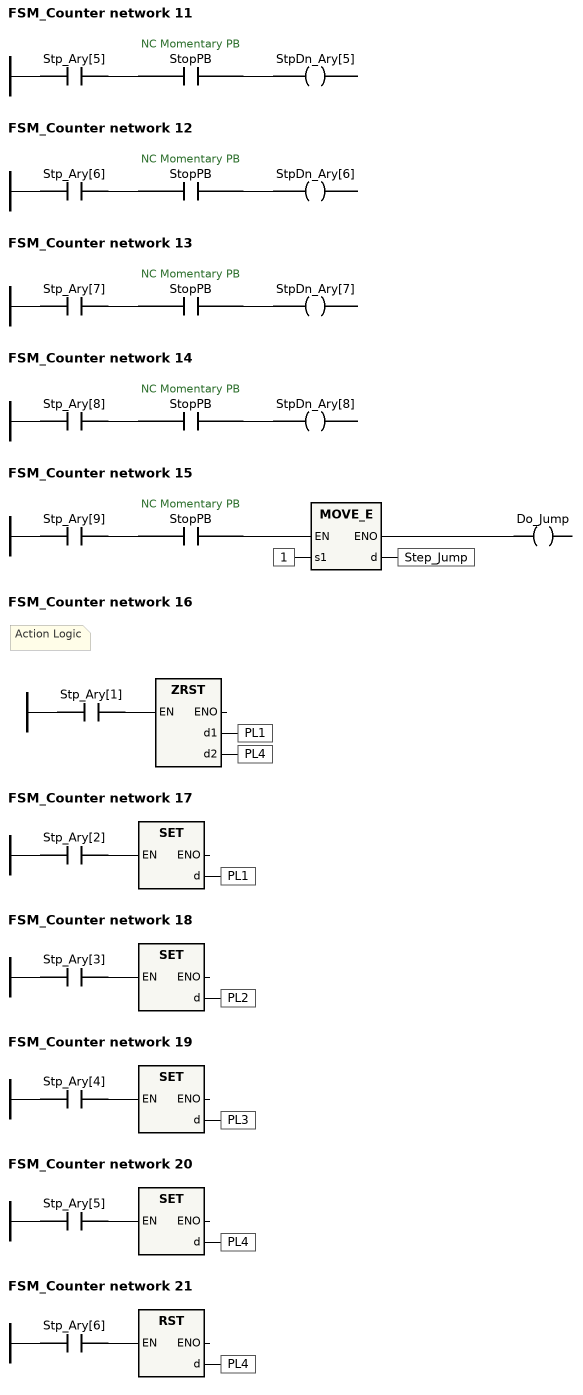
(* network 11 *)
StpDn_Ary[5] := Stp_Ary[5] AND StopPB;
(* network 12 *)
StpDn_Ary[6] := Stp_Ary[6] AND StopPB;
(* network 13 *)
StpDn_Ary[7] := Stp_Ary[7] AND StopPB;
(* network 14 *)
StpDn_Ary[8] := Stp_Ary[8] AND StopPB;
(* network 15 *)
_e1 := MOVE_E(Stp_Ary[9] AND StopPB, 1, Step_Jump);
Do_Jump := _e1;
(* network 16 *)
(* Action Logic *)
ZRST(Stp_Ary[1], PL1, PL4);
(* network 17 *)
SET(Stp_Ary[2], PL1);
(* network 18 *)
SET(Stp_Ary[3], PL2);
(* network 19 *)
SET(Stp_Ary[4], PL3);
(* network 20 *)
SET(Stp_Ary[5], PL4);
(* network 21 *)
RST(Stp_Ary[6], PL4);
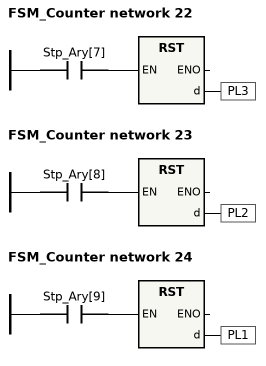
(* network 22 *)
RST(Stp_Ary[7], PL3);
(* network 23 *)
RST(Stp_Ary[8], PL2);
(* network 24 *)
RST(Stp_Ary[9], PL1);
END_PROGRAM

FUNCTION_BLOCK Get_Step_D
VAR_OUTPUT
  GSOut : BOOL;
END_VAR
VAR_IN_OUT
  SArray : ARRAY [0..15] OF BOOL;
END_VAR
VAR_INPUT
  StpNum : INT;
END_VAR
GSOut := SArray[StpNum];
END_FUNCTION_BLOCK

FUNCTION_BLOCK SR_Step_D
VAR_INPUT
  In : BOOL;
  StpNum : INT;
END_VAR
VAR_IN_OUT
  SArray : ARRAY [0..15] OF BOOL;
END_VAR
SArray[StpNum] := In;
END_FUNCTION_BLOCK

PROGRAM FSM_Counter_D
VAR
  StepCtrCV : INT;
  ClrStep : SR_Step;
  SetStep : SR_Step;
  Reset : BOOL;
  Do_Jump : BOOL;
  Step_Jump : INT;
  R_TRIG_1 : R_TRIG;
  Get_Step_D_1 : Get_Step_D;
  SR_Step_D_1 : SR_Step_D;
  SR_Step_D_2 : SR_Step_D;
END_VAR
(* structured ladder/FBD written out as ST: instructions are called as NAME(EN, inputs, outputs); _pN, _eN, _tN stand for wires *)
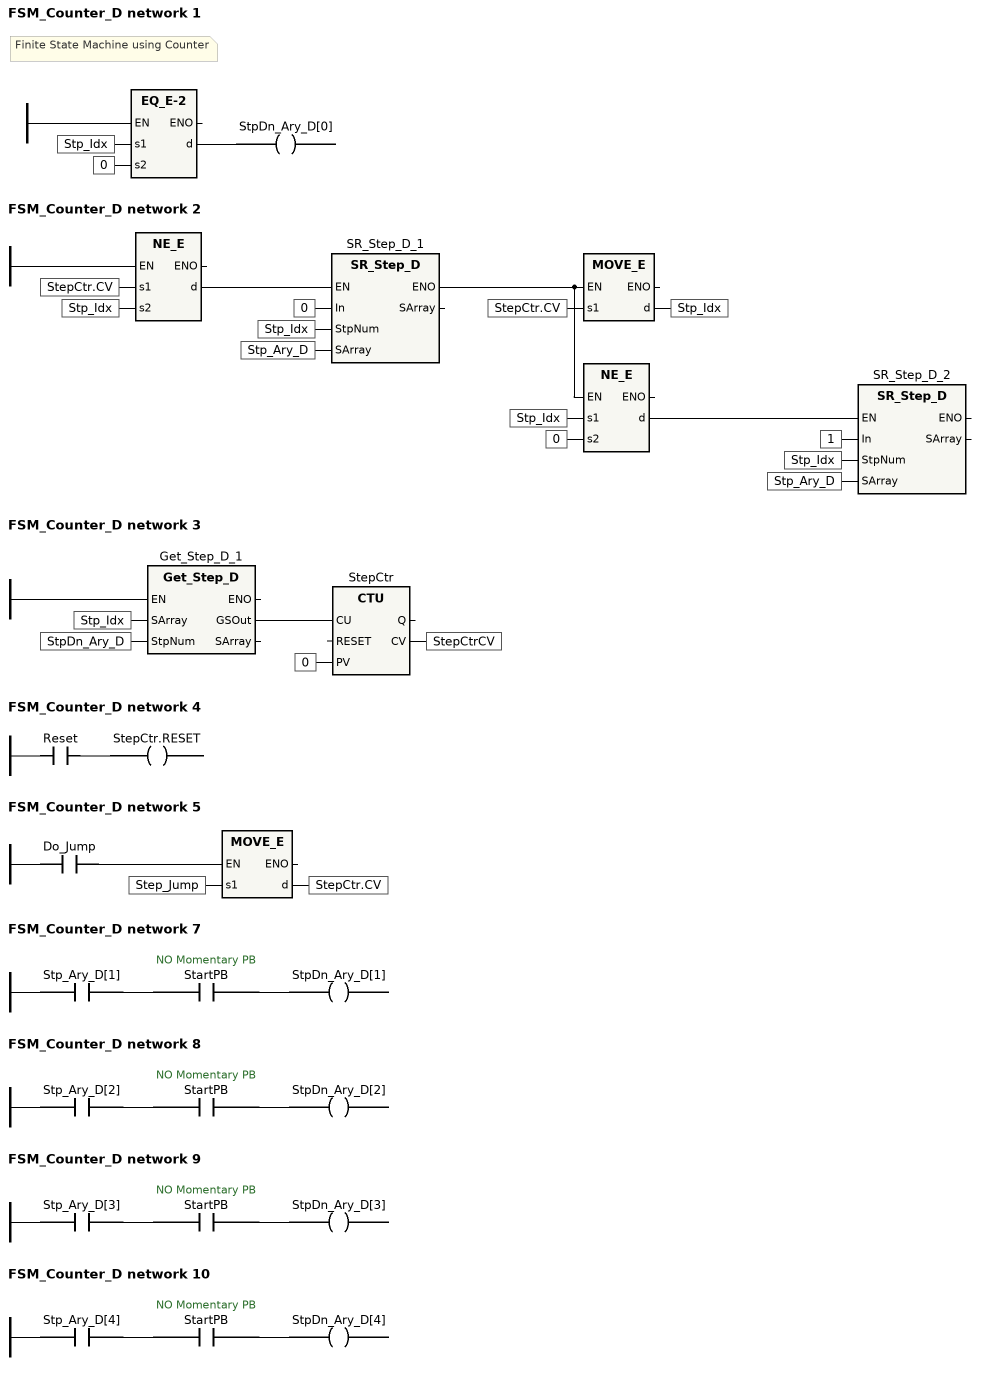
(* network 1 *)
(* Finite State Machine using Counter *)
EQ_E(TRUE, Stp_Idx, 0, _t1);
StpDn_Ary_D[0] := _t1;
(* network 2 *)
NE_E(TRUE, StepCtr.CV, Stp_Idx, _t1);
SR_Step_D_1(EN := _t1, In := 0, StpNum := Stp_Idx, SArray := Stp_Ary_D);
MOVE_E(SR_Step_D_1.ENO, StepCtr.CV, Stp_Idx);
NE_E(SR_Step_D_1.ENO, Stp_Idx, 0, _t2);
SR_Step_D_2(EN := _t2, In := 1, StpNum := Stp_Idx, SArray := Stp_Ary_D);
(* network 3 *)
Get_Step_D_1(EN := TRUE, SArray := Stp_Idx, StpNum := StpDn_Ary_D);
StepCtr(CU := Get_Step_D_1.GSOut, PV := 0, CV => StepCtrCV);
(* network 4 *)
StepCtr.RESET := Reset;
(* network 5 *)
MOVE_E(Do_Jump, Step_Jump, StepCtr.CV);
(* Transition Logic *)
(* network 7 *)
StpDn_Ary_D[1] := Stp_Ary_D[1] AND StartPB;
(* network 8 *)
StpDn_Ary_D[2] := Stp_Ary_D[2] AND StartPB;
(* network 9 *)
StpDn_Ary_D[3] := Stp_Ary_D[3] AND StartPB;
(* network 10 *)
StpDn_Ary_D[4] := Stp_Ary_D[4] AND StartPB;
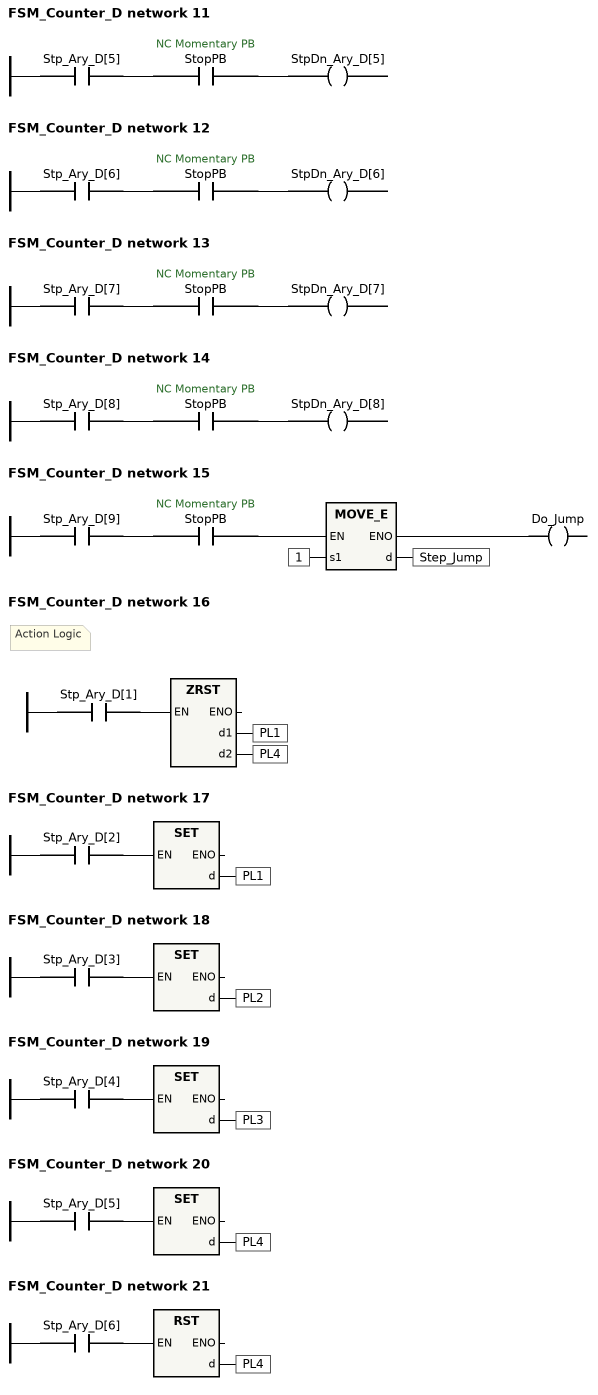
(* network 11 *)
StpDn_Ary_D[5] := Stp_Ary_D[5] AND StopPB;
(* network 12 *)
StpDn_Ary_D[6] := Stp_Ary_D[6] AND StopPB;
(* network 13 *)
StpDn_Ary_D[7] := Stp_Ary_D[7] AND StopPB;
(* network 14 *)
StpDn_Ary_D[8] := Stp_Ary_D[8] AND StopPB;
(* network 15 *)
_e1 := MOVE_E(Stp_Ary_D[9] AND StopPB, 1, Step_Jump);
Do_Jump := _e1;
(* network 16 *)
(* Action Logic *)
ZRST(Stp_Ary_D[1], PL1, PL4);
(* network 17 *)
SET(Stp_Ary_D[2], PL1);
(* network 18 *)
SET(Stp_Ary_D[3], PL2);
(* network 19 *)
SET(Stp_Ary_D[4], PL3);
(* network 20 *)
SET(Stp_Ary_D[5], PL4);
(* network 21 *)
RST(Stp_Ary_D[6], PL4);
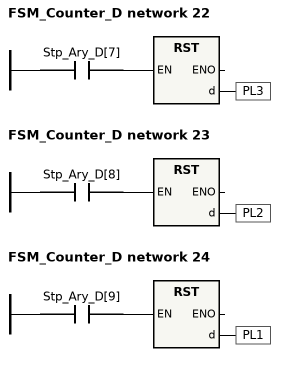
(* network 22 *)
RST(Stp_Ary_D[7], PL3);
(* network 23 *)
RST(Stp_Ary_D[8], PL2);
(* network 24 *)
RST(Stp_Ary_D[9], PL1);
END_PROGRAM

PROGRAM FSM_EQU2
(* structured ladder/FBD written out as ST: instructions are called as NAME(EN, inputs, outputs); _pN, _eN, _tN stand for wires *)
(* Instructions Supported in Simulator and LE3U Trainer *)
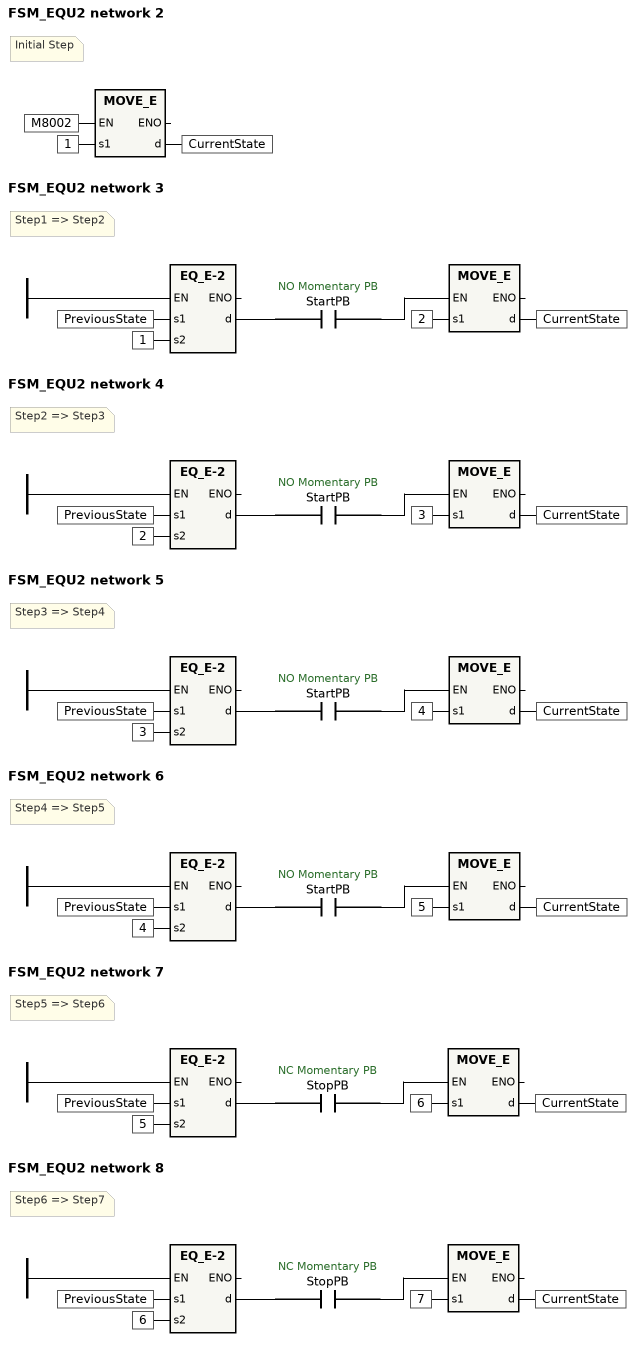
(* network 2 *)
(* Initial Step *)
MOVE_E(M8002, 1, CurrentState);
(* network 3 *)
(* Step1 => Step2 *)
EQ_E(TRUE, PreviousState, 1, _t1);
MOVE_E(_t1 AND StartPB, 2, CurrentState);
(* network 4 *)
(* Step2 => Step3 *)
EQ_E(TRUE, PreviousState, 2, _t1);
MOVE_E(_t1 AND StartPB, 3, CurrentState);
(* network 5 *)
(* Step3 => Step4 *)
EQ_E(TRUE, PreviousState, 3, _t1);
MOVE_E(_t1 AND StartPB, 4, CurrentState);
(* network 6 *)
(* Step4 => Step5 *)
EQ_E(TRUE, PreviousState, 4, _t1);
MOVE_E(_t1 AND StartPB, 5, CurrentState);
(* network 7 *)
(* Step5 => Step6 *)
EQ_E(TRUE, PreviousState, 5, _t1);
MOVE_E(_t1 AND StopPB, 6, CurrentState);
(* network 8 *)
(* Step6 => Step7 *)
EQ_E(TRUE, PreviousState, 6, _t1);
MOVE_E(_t1 AND StopPB, 7, CurrentState);
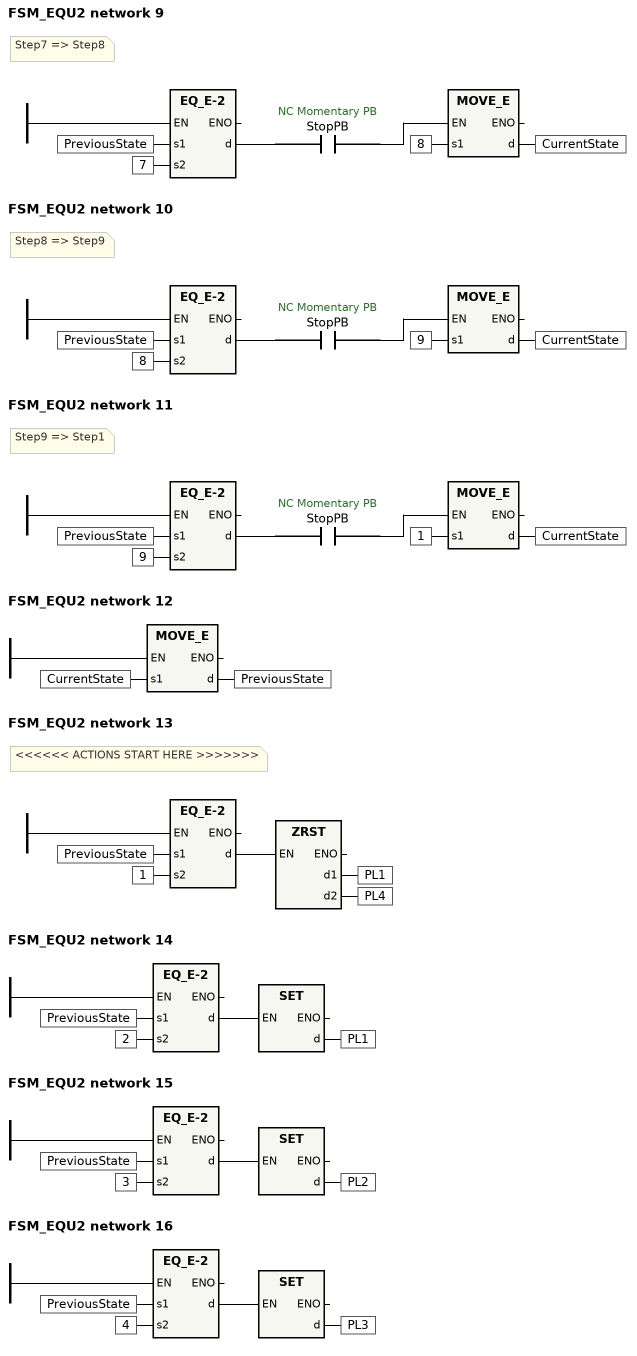
(* network 9 *)
(* Step7 => Step8 *)
EQ_E(TRUE, PreviousState, 7, _t1);
MOVE_E(_t1 AND StopPB, 8, CurrentState);
(* network 10 *)
(* Step8 => Step9 *)
EQ_E(TRUE, PreviousState, 8, _t1);
MOVE_E(_t1 AND StopPB, 9, CurrentState);
(* network 11 *)
(* Step9 => Step1 *)
EQ_E(TRUE, PreviousState, 9, _t1);
MOVE_E(_t1 AND StopPB, 1, CurrentState);
(* network 12 *)
MOVE_E(TRUE, CurrentState, PreviousState);
(* network 13 *)
(* <<<<<< ACTIONS START HERE >>>>>>> *)
EQ_E(TRUE, PreviousState, 1, _t1);
ZRST(_t1, PL1, PL4);
(* network 14 *)
EQ_E(TRUE, PreviousState, 2, _t1);
SET(_t1, PL1);
(* network 15 *)
EQ_E(TRUE, PreviousState, 3, _t1);
SET(_t1, PL2);
(* network 16 *)
EQ_E(TRUE, PreviousState, 4, _t1);
SET(_t1, PL3);
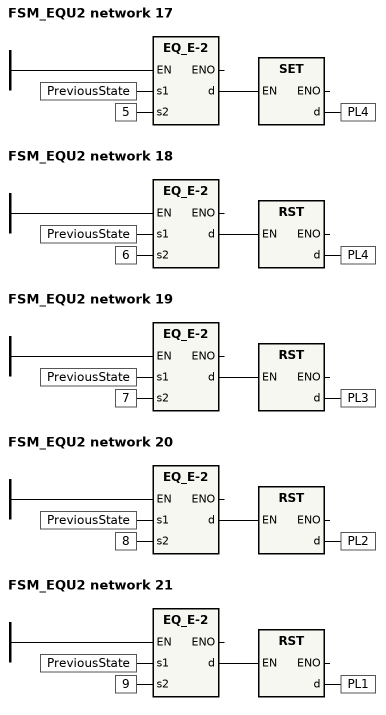
(* network 17 *)
EQ_E(TRUE, PreviousState, 5, _t1);
SET(_t1, PL4);
(* network 18 *)
EQ_E(TRUE, PreviousState, 6, _t1);
RST(_t1, PL4);
(* network 19 *)
EQ_E(TRUE, PreviousState, 7, _t1);
RST(_t1, PL3);
(* network 20 *)
EQ_E(TRUE, PreviousState, 8, _t1);
RST(_t1, PL2);
(* network 21 *)
EQ_E(TRUE, PreviousState, 9, _t1);
RST(_t1, PL1);
END_PROGRAM

// device comments not shown above
M8000  ; Always On
M8002  ; First Scan
C0  ; StpCounter
